(* CODESYS project proj_12_18_zad1.project

Project tree, tasks and I/O mapping:
  Device : Berghof MX6 Control, Berghof Automation GmbH, version 1.8.0.0
    application Application
      libraries: Standard, * (System)
      task MainTask (cyclic, interval t#25ms, priority 1) calls PLC_PRG
      program PLC_PRG [LD]
      visualisation Visualization
      function F_KIERUNEK [LD]
      function block FB_TIMERY [LD]
      function block FB_STER_NAPEDU [LD]
    Extension_Slots : Extension Slots, Berghof Automation GmbH, version 1.2.0.3
      XBIO_Berghof_IO : XBIO Berghof IO, Berghof Automation GmbH, version 1.2.0.3
          unmapped channels: Digital Input 0, Digital Input 1, Digital Input 2, Digital Input 3, Digital Input 4, Digital Output 0, Digital Output 1, Digital Output 2, Digital Output 3, Digital Output 4, Channel 0, Channel 1, Channel 2, Channel 3, Channel 4, Channel 5, Channel 6, Channel 7, Channel 8, Channel 9, Channel 10, Channel 11, Channel 0, Channel 1, Channel 2, Channel 3, Channel 4, Channel 5, Channel 6, Channel 7, Counter/Encoder 0, Counter/Encoder 1, Differential Counter/Encoder (0+1), DUMMY 0
      <Empty>
  text list GlobalTextList
  function block FB_STER_NAPEDU [LD]
*)

// Device/Application/PLC_PRG
PROGRAM PLC_PRG
VAR_INPUT
	CWL AT %IX0.0: BOOL;
	CWLP AT %IX0.1: BOOL;
	CWP AT %IX0.2: BOOL;
	CWPP AT %IX0.3: BOOL;
	TRASA AT %IX0.4: BOOL;
END_VAR
VAR_OUTPUT
	POD_1 AT %QX0.0: BOOL;
	POD_2 AT %QX0.1: BOOL;
	POD_3L AT %QX0.2: BOOL;
	POD_3P AT %QX0.3: BOOL;
	K1 AT %QX0.4: BOOL;
	K2 AT %QX0.5: BOOL;
END_VAR
VAR
	LICZ: CTU;
	NUM: WORD;
	FB_TIMERY_0: FB_TIMERY;
	FB_STER_NAPEDU: FB_STER_NAPEDU;
	TON1: TON;
	T1: TIME;
	FB_STER_NAPEDU_P1: FB_STER_NAPEDU;
	FB_STER_NAPEDU_P2: FB_STER_NAPEDU;
END_VAR
VAR_INPUT
	CT_RES AT %IX0.5: BOOL;
END_VAR
VAR_OUTPUT
	CT_OUT: BOOL;
END_VAR

VAR_INPUT
	ZAL_WYL_AUT_IN: BOOL;
	PRAWO_LEWO_AUT_IN: BOOL;
	ZAL_WYL_LOK_IN: BOOL;
	PRAWO_LEWO_LOK_IN: BOOL;
	POTW_ROZR_IN: BOOL;
	BLAD_ASYM_IN: BOOL;
	BLAD_TEMP_IN: BOOL;
	CHCE_LOK_IN: BOOL;
	POTW_LOK_IN: BOOL;
END_VAR

VAR_OUTPUT
	ZAL_WYL_OUT: BOOL;
	PRAWO_LEWO_OUT: BOOL;
	SYGN_OSTRZ_OUT: BOOL;
	BLAD_OUT: BOOL;
	CHCE_LOK_OUT: BOOL;
	LOK_OUT: BOOL;
	AUT_OUT: BOOL;
END_VAR
VAR_INPUT
	KASOWANIE_ALARMU: BOOL;
END_VAR
VAR
	TON0: TON;
	T0: TIME;
END_VAR
VAR_OUTPUT
	ZAL_WYL_OUT_P1: BOOL;
	ZAL_WYL_OUT_P2: BOOL;
	SYGN_OSTRZ_OUT_P1: BOOL;
	SYGN_OSTRZ_OUT_P2: BOOL;
	BLAD_OUT_P1: BOOL;
	BLAD_OUT_P2: BOOL;
	CHCE_LOK_OUT_P1: BOOL;
	CHCE_LOK_OUT_P2: BOOL;
	LOK_OUT_P1: BOOL;
	LOK_OUT_P2: BOOL;
	AUT_OUT_P1: BOOL;
	AUT_OUT_P2: BOOL;
END_VAR
VAR_INPUT
	ZAL_WYL_LOK_IN_P1: BOOL;
	ZAL_WYL_LOK_IN_P2: BOOL;
	POTW_ROZR_IN_P1: BOOL;
	POTW_ROZR_IN_P2: BOOL;
	BLAD_ASYM_IN_P1: BOOL;
	BLAD_ASYM_IN_P2: BOOL;
	BLAD_TEMP_IN_P1: BOOL;
	BLAD_TEMP_IN_P2: BOOL;
	CHCE_LOK_IN_P1: BOOL;
	CHCE_LOK_IN_P2: BOOL;
	POTW_LOK_IN_P1: BOOL;
	POTW_LOK_IN_P2: BOOL;
END_VAR
VAR
	M1: BOOL;
	M2: BOOL;
END_VAR

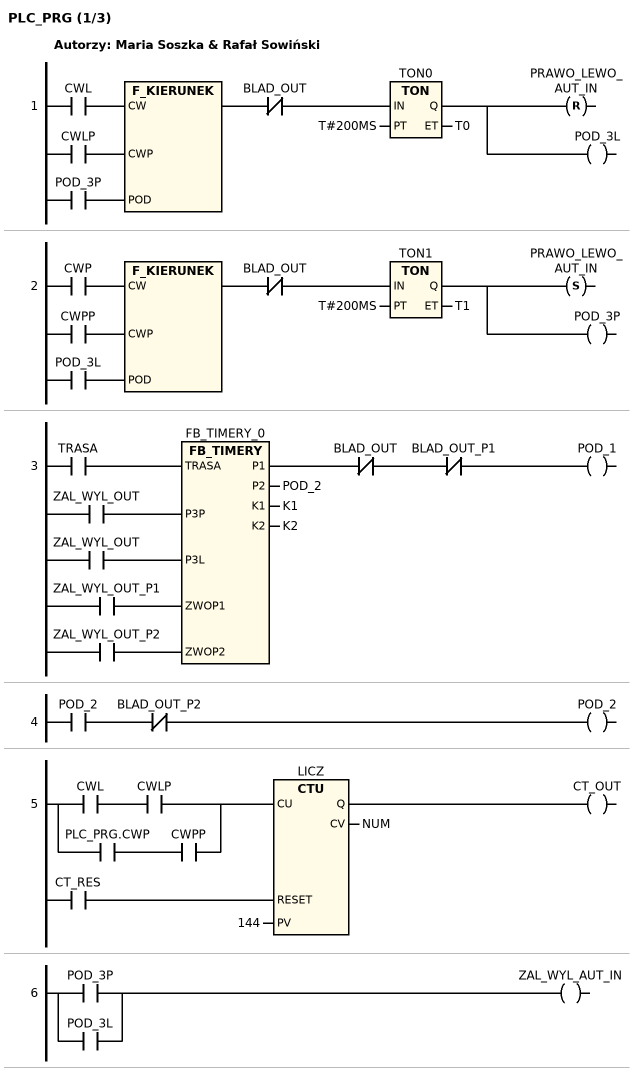
// NETWORK 1: Autorzy: Maria Soszka & Rafał Sowiński
TON0(IN := F_KIERUNEK(CW := CWL, CWP := CWLP, POD := POD_3P) AND NOT BLAD_OUT, PT := T#200MS, ET => T0); // TON
PRAWO_LEWO_AUT_IN R= TON0.Q;
POD_3L := TON0.Q;

// NETWORK 2
TON1(IN := F_KIERUNEK(CW := CWP, CWP := CWPP, POD := POD_3L) AND NOT BLAD_OUT, PT := T#200MS, ET => T1); // TON
PRAWO_LEWO_AUT_IN S= TON1.Q;
POD_3P := TON1.Q;

// NETWORK 3
FB_TIMERY_0(
    TRASA := TRASA,
    P3P := ZAL_WYL_OUT,
    P3L := ZAL_WYL_OUT,
    ZWOP1 := ZAL_WYL_OUT_P1,
    ZWOP2 := ZAL_WYL_OUT_P2,
    P2 => POD_2,
    K1 => K1,
    K2 => K2); // FB_TIMERY
POD_1 := FB_TIMERY_0.P1 AND NOT BLAD_OUT AND NOT BLAD_OUT_P1;

// NETWORK 4
POD_2 := POD_2 AND NOT BLAD_OUT_P2;

// NETWORK 5
LICZ(CU := CWL AND CWLP OR PLC_PRG.CWP AND CWPP, RESET := CT_RES, PV := 144, CV => NUM); // CTU
CT_OUT := LICZ.Q;

// NETWORK 6
ZAL_WYL_AUT_IN := POD_3P OR POD_3L;

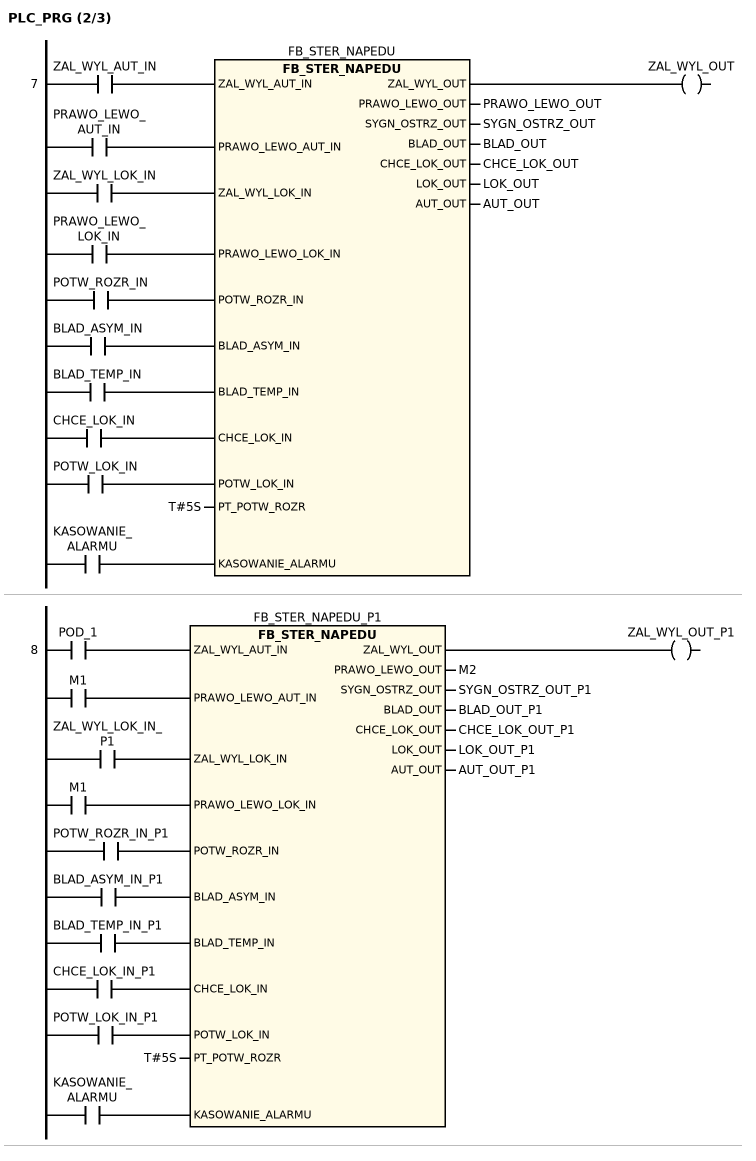
// NETWORK 7
FB_STER_NAPEDU(
    ZAL_WYL_AUT_IN := ZAL_WYL_AUT_IN,
    PRAWO_LEWO_AUT_IN := PRAWO_LEWO_AUT_IN,
    ZAL_WYL_LOK_IN := ZAL_WYL_LOK_IN,
    PRAWO_LEWO_LOK_IN := PRAWO_LEWO_LOK_IN,
    POTW_ROZR_IN := POTW_ROZR_IN,
    BLAD_ASYM_IN := BLAD_ASYM_IN,
    BLAD_TEMP_IN := BLAD_TEMP_IN,
    CHCE_LOK_IN := CHCE_LOK_IN,
    POTW_LOK_IN := POTW_LOK_IN,
    PT_POTW_ROZR := T#5S,
    KASOWANIE_ALARMU := KASOWANIE_ALARMU,
    PRAWO_LEWO_OUT => PRAWO_LEWO_OUT,
    SYGN_OSTRZ_OUT => SYGN_OSTRZ_OUT,
    BLAD_OUT => BLAD_OUT,
    CHCE_LOK_OUT => CHCE_LOK_OUT,
    LOK_OUT => LOK_OUT,
    AUT_OUT => AUT_OUT);
ZAL_WYL_OUT := FB_STER_NAPEDU.ZAL_WYL_OUT;

// NETWORK 8
FB_STER_NAPEDU_P1(
    ZAL_WYL_AUT_IN := POD_1,
    PRAWO_LEWO_AUT_IN := M1,
    ZAL_WYL_LOK_IN := ZAL_WYL_LOK_IN_P1,
    PRAWO_LEWO_LOK_IN := M1,
    POTW_ROZR_IN := POTW_ROZR_IN_P1,
    BLAD_ASYM_IN := BLAD_ASYM_IN_P1,
    BLAD_TEMP_IN := BLAD_TEMP_IN_P1,
    CHCE_LOK_IN := CHCE_LOK_IN_P1,
    POTW_LOK_IN := POTW_LOK_IN_P1,
    PT_POTW_ROZR := T#5S,
    KASOWANIE_ALARMU := KASOWANIE_ALARMU,
    PRAWO_LEWO_OUT => M2,
    SYGN_OSTRZ_OUT => SYGN_OSTRZ_OUT_P1,
    BLAD_OUT => BLAD_OUT_P1,
    CHCE_LOK_OUT => CHCE_LOK_OUT_P1,
    LOK_OUT => LOK_OUT_P1,
    AUT_OUT => AUT_OUT_P1); // FB_STER_NAPEDU
ZAL_WYL_OUT_P1 := FB_STER_NAPEDU_P1.ZAL_WYL_OUT;

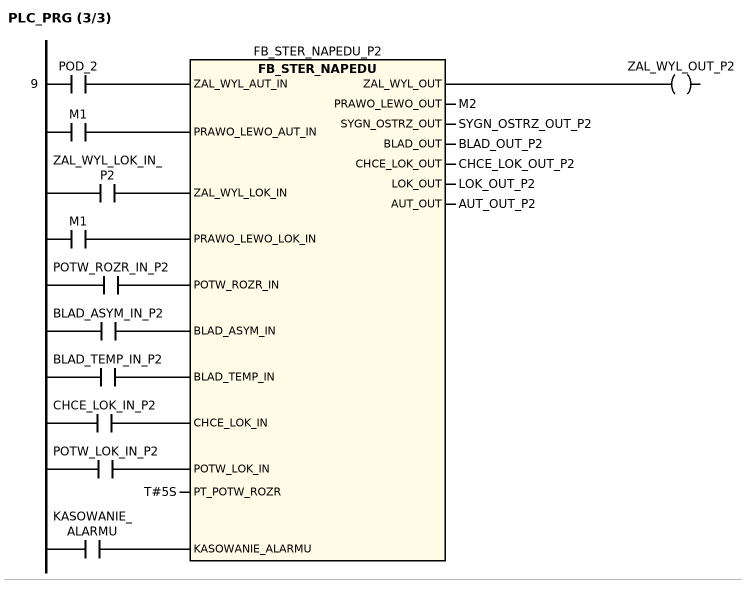
// NETWORK 9
FB_STER_NAPEDU_P2(
    ZAL_WYL_AUT_IN := POD_2,
    PRAWO_LEWO_AUT_IN := M1,
    ZAL_WYL_LOK_IN := ZAL_WYL_LOK_IN_P2,
    PRAWO_LEWO_LOK_IN := M1,
    POTW_ROZR_IN := POTW_ROZR_IN_P2,
    BLAD_ASYM_IN := BLAD_ASYM_IN_P2,
    BLAD_TEMP_IN := BLAD_TEMP_IN_P2,
    CHCE_LOK_IN := CHCE_LOK_IN_P2,
    POTW_LOK_IN := POTW_LOK_IN_P2,
    PT_POTW_ROZR := T#5S,
    KASOWANIE_ALARMU := KASOWANIE_ALARMU,
    PRAWO_LEWO_OUT => M2,
    SYGN_OSTRZ_OUT => SYGN_OSTRZ_OUT_P2,
    BLAD_OUT => BLAD_OUT_P2,
    CHCE_LOK_OUT => CHCE_LOK_OUT_P2,
    LOK_OUT => LOK_OUT_P2,
    AUT_OUT => AUT_OUT_P2); // FB_STER_NAPEDU
ZAL_WYL_OUT_P2 := FB_STER_NAPEDU_P2.ZAL_WYL_OUT;

END_PROGRAM

// Device/Application/F_KIERUNEK
FUNCTION F_KIERUNEK : BOOL
VAR_INPUT
	CW: BOOL;
	CWP: BOOL;
	POD: BOOL;
END_VAR

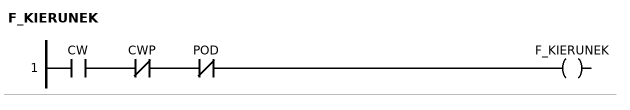
// NETWORK 1
F_KIERUNEK := CW AND NOT CWP AND NOT POD;

END_FUNCTION

// Device/Application/FB_TIMERY
FUNCTION_BLOCK FB_TIMERY
VAR_INPUT
	TRASA: BOOL;
END_VAR
VAR_OUTPUT
	P1: BOOL;
	P2: BOOL;
	K1: BOOL;
	K2: BOOL;
END_VAR
VAR
	TIM1: TON;
	T1: TIME;
	TIM2: TON;
	T2: TIME;
	TIMK1: TON;
	TIMK2: TON;
	TK1: TIME;
	TK2: TIME;
END_VAR
VAR_INPUT
	P3P: BOOL;
	P3L: BOOL;
	ZWOP1: BOOL;
	ZWOP2: BOOL;
END_VAR
VAR // added by the converter: edge detectors and wires of the graphical bodies
    _w1 : BOOL;
END_VAR

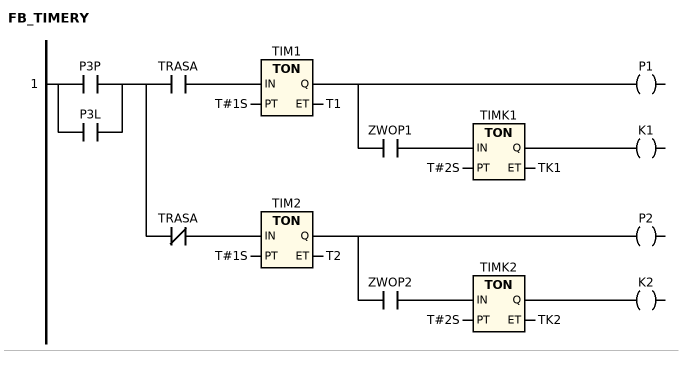
// NETWORK 1
_w1 := P3P OR P3L;
TIM1(IN := _w1 AND TRASA, PT := T#1S, ET => T1); // TON
P1 := TIM1.Q;
TIMK1(IN := TIM1.Q AND ZWOP1, PT := T#2S, ET => TK1); // TON
K1 := TIMK1.Q;
TIM2(IN := _w1 AND NOT TRASA, PT := T#1S, ET => T2); // TON
P2 := TIM2.Q;
TIMK2(IN := TIM2.Q AND ZWOP2, PT := T#2S, ET => TK2); // TON
K2 := TIMK2.Q;

END_FUNCTION_BLOCK

// FB_STER_NAPEDU
FUNCTION_BLOCK FB_STER_NAPEDU
VAR_INPUT
	ZAL_WYL_AUT_IN: BOOL;
	PRAWO_LEWO_AUT_IN: BOOL;
	ZAL_WYL_LOK_IN: BOOL;
	PRAWO_LEWO_LOK_IN: BOOL;
	POTW_ROZR_IN: BOOL;
	BLAD_ASYM_IN: BOOL;
	BLAD_TEMP_IN: BOOL;
	CHCE_LOK_IN: BOOL;
	POTW_LOK_IN: BOOL;
END_VAR
VAR_OUTPUT
	ZAL_WYL_OUT: BOOL;
	PRAWO_LEWO_OUT: BOOL;
	SYGN_OSTRZ_OUT: BOOL;
	BLAD_OUT: BOOL;
	CHCE_LOK_OUT: BOOL;
	LOK_OUT: BOOL;
	AUT_OUT: BOOL;
END_VAR
VAR
	BRAK_POTW_ROZR: BOOL;
	TON_SYGN_OSTRZ: TON;
	T_SYGN_OSTRZ: TIME;
	PT_SYGN_OSTRZ: TIME := T#3S;
	TON_POTW_ROZR: TON;
	T_POTW_ROZR: TIME;
END_VAR
VAR_INPUT
	PT_POTW_ROZR: TIME;
END_VAR
VAR // added by the converter: edge detectors and wires of the graphical bodies
    _w1 : BOOL;
END_VAR

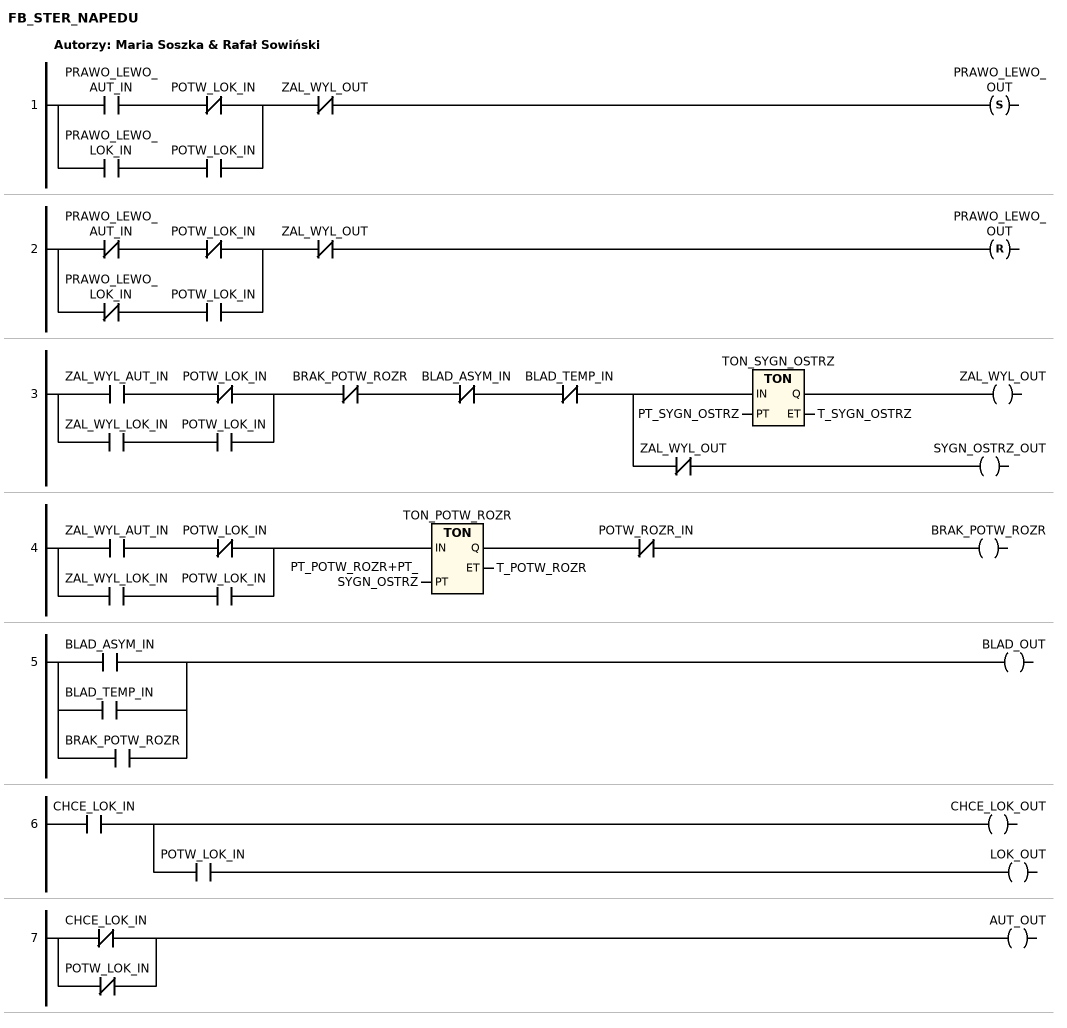
// NETWORK 1: Autorzy: Maria Soszka & Rafał Sowiński
PRAWO_LEWO_OUT S= (PRAWO_LEWO_AUT_IN AND NOT POTW_LOK_IN OR PRAWO_LEWO_LOK_IN AND POTW_LOK_IN) AND NOT ZAL_WYL_OUT;

// NETWORK 2
PRAWO_LEWO_OUT R= (NOT PRAWO_LEWO_AUT_IN AND NOT POTW_LOK_IN OR NOT PRAWO_LEWO_LOK_IN AND POTW_LOK_IN) AND NOT ZAL_WYL_OUT;

// NETWORK 3
_w1 := (ZAL_WYL_AUT_IN AND NOT POTW_LOK_IN OR ZAL_WYL_LOK_IN AND POTW_LOK_IN) AND NOT BRAK_POTW_ROZR AND NOT BLAD_ASYM_IN AND NOT BLAD_TEMP_IN;
TON_SYGN_OSTRZ(IN := _w1, PT := PT_SYGN_OSTRZ, ET => T_SYGN_OSTRZ); // TON
ZAL_WYL_OUT := TON_SYGN_OSTRZ.Q;
SYGN_OSTRZ_OUT := _w1 AND NOT ZAL_WYL_OUT;

// NETWORK 4
TON_POTW_ROZR(
    IN := ZAL_WYL_AUT_IN AND NOT POTW_LOK_IN OR ZAL_WYL_LOK_IN AND POTW_LOK_IN,
    PT := PT_POTW_ROZR+PT_SYGN_OSTRZ,
    ET => T_POTW_ROZR); // TON
BRAK_POTW_ROZR := TON_POTW_ROZR.Q AND NOT POTW_ROZR_IN;

// NETWORK 5
BLAD_OUT := BLAD_ASYM_IN OR BLAD_TEMP_IN OR BRAK_POTW_ROZR;

// NETWORK 6
CHCE_LOK_OUT := CHCE_LOK_IN;
LOK_OUT := CHCE_LOK_IN AND POTW_LOK_IN;

// NETWORK 7
AUT_OUT := NOT CHCE_LOK_IN OR NOT POTW_LOK_IN;

END_FUNCTION_BLOCK

// Device/Application/FB_STER_NAPEDU
FUNCTION_BLOCK FB_STER_NAPEDU
VAR_INPUT
	ZAL_WYL_AUT_IN: BOOL;
	PRAWO_LEWO_AUT_IN: BOOL;
	ZAL_WYL_LOK_IN: BOOL;
	PRAWO_LEWO_LOK_IN: BOOL;
	POTW_ROZR_IN: BOOL;
	BLAD_ASYM_IN: BOOL;
	BLAD_TEMP_IN: BOOL;
	CHCE_LOK_IN: BOOL;
	POTW_LOK_IN: BOOL;
END_VAR
VAR_OUTPUT
	ZAL_WYL_OUT: BOOL;
	PRAWO_LEWO_OUT: BOOL;
	SYGN_OSTRZ_OUT: BOOL;
	BLAD_OUT: BOOL;
	CHCE_LOK_OUT: BOOL;
	LOK_OUT: BOOL;
	AUT_OUT: BOOL;
END_VAR
VAR
	BRAK_POTW_ROZR: BOOL;
	TON_SYGN_OSTRZ: TON;
	T_SYGN_OSTRZ: TIME;
	PT_SYGN_OSTRZ: TIME := T#3S;
	TON_POTW_ROZR: TON;
	T_POTW_ROZR: TIME;
END_VAR
VAR_INPUT
	PT_POTW_ROZR: TIME;
	KASOWANIE_ALARMU: BOOL;
END_VAR
VAR // added by the converter: edge detectors and wires of the graphical bodies
    _w1 : BOOL;
END_VAR

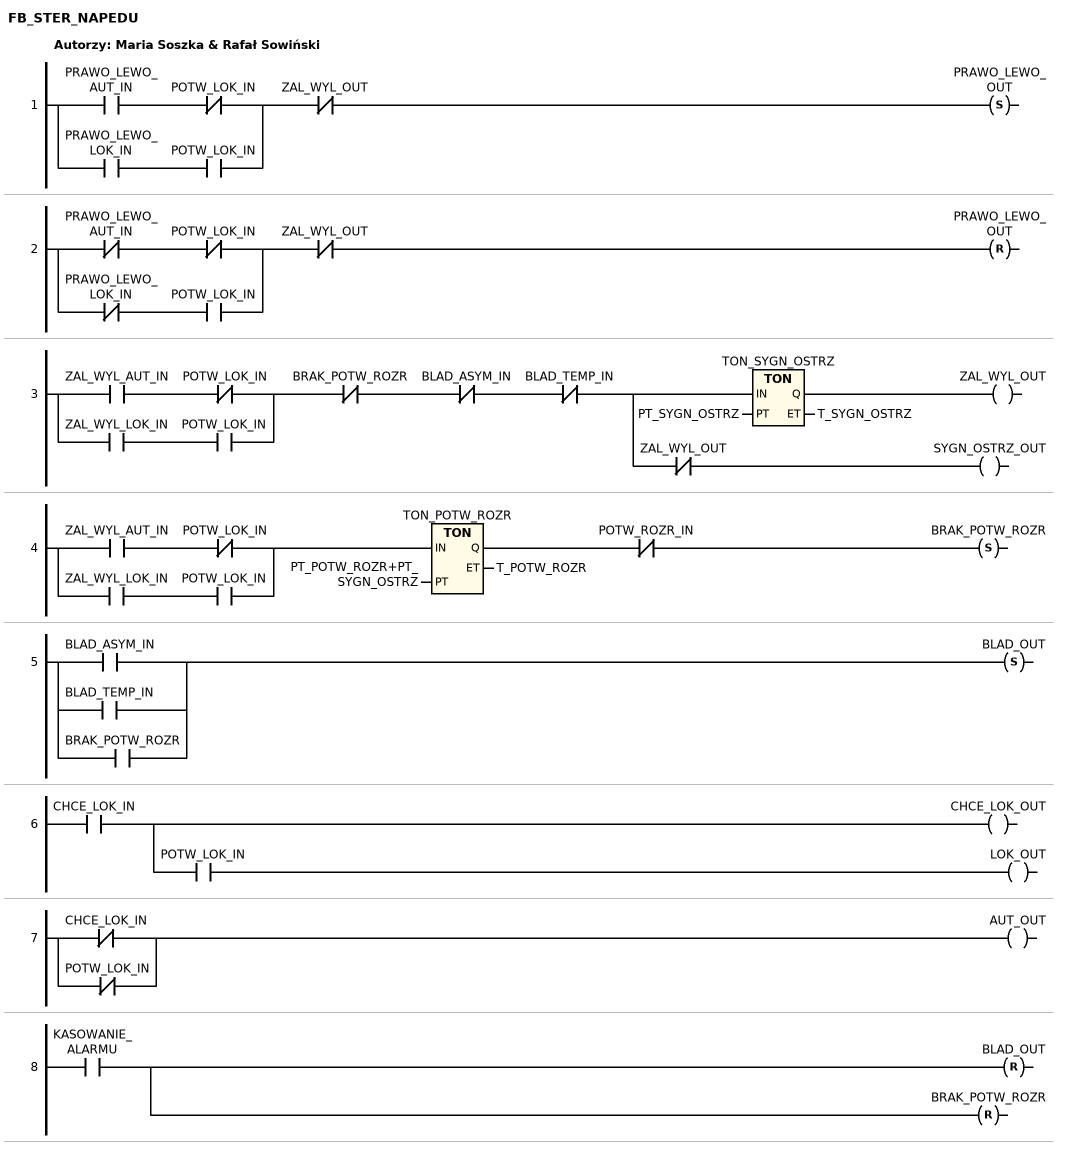
// NETWORK 1: Autorzy: Maria Soszka & Rafał Sowiński
PRAWO_LEWO_OUT S= (PRAWO_LEWO_AUT_IN AND NOT POTW_LOK_IN OR PRAWO_LEWO_LOK_IN AND POTW_LOK_IN) AND NOT ZAL_WYL_OUT;

// NETWORK 2
PRAWO_LEWO_OUT R= (NOT PRAWO_LEWO_AUT_IN AND NOT POTW_LOK_IN OR NOT PRAWO_LEWO_LOK_IN AND POTW_LOK_IN) AND NOT ZAL_WYL_OUT;

// NETWORK 3
_w1 := (ZAL_WYL_AUT_IN AND NOT POTW_LOK_IN OR ZAL_WYL_LOK_IN AND POTW_LOK_IN) AND NOT BRAK_POTW_ROZR AND NOT BLAD_ASYM_IN AND NOT BLAD_TEMP_IN;
TON_SYGN_OSTRZ(IN := _w1, PT := PT_SYGN_OSTRZ, ET => T_SYGN_OSTRZ); // TON
ZAL_WYL_OUT := TON_SYGN_OSTRZ.Q;
SYGN_OSTRZ_OUT := _w1 AND NOT ZAL_WYL_OUT;

// NETWORK 4
TON_POTW_ROZR(
    IN := ZAL_WYL_AUT_IN AND NOT POTW_LOK_IN OR ZAL_WYL_LOK_IN AND POTW_LOK_IN,
    PT := PT_POTW_ROZR+PT_SYGN_OSTRZ,
    ET => T_POTW_ROZR); // TON
BRAK_POTW_ROZR S= TON_POTW_ROZR.Q AND NOT POTW_ROZR_IN;

// NETWORK 5
BLAD_OUT S= BLAD_ASYM_IN OR BLAD_TEMP_IN OR BRAK_POTW_ROZR;

// NETWORK 6
CHCE_LOK_OUT := CHCE_LOK_IN;
LOK_OUT := CHCE_LOK_IN AND POTW_LOK_IN;

// NETWORK 7
AUT_OUT := NOT CHCE_LOK_IN OR NOT POTW_LOK_IN;

// NETWORK 8
BLAD_OUT R= KASOWANIE_ALARMU;
BRAK_POTW_ROZR R= KASOWANIE_ALARMU;

END_FUNCTION_BLOCK

// Device/Application/Visualization
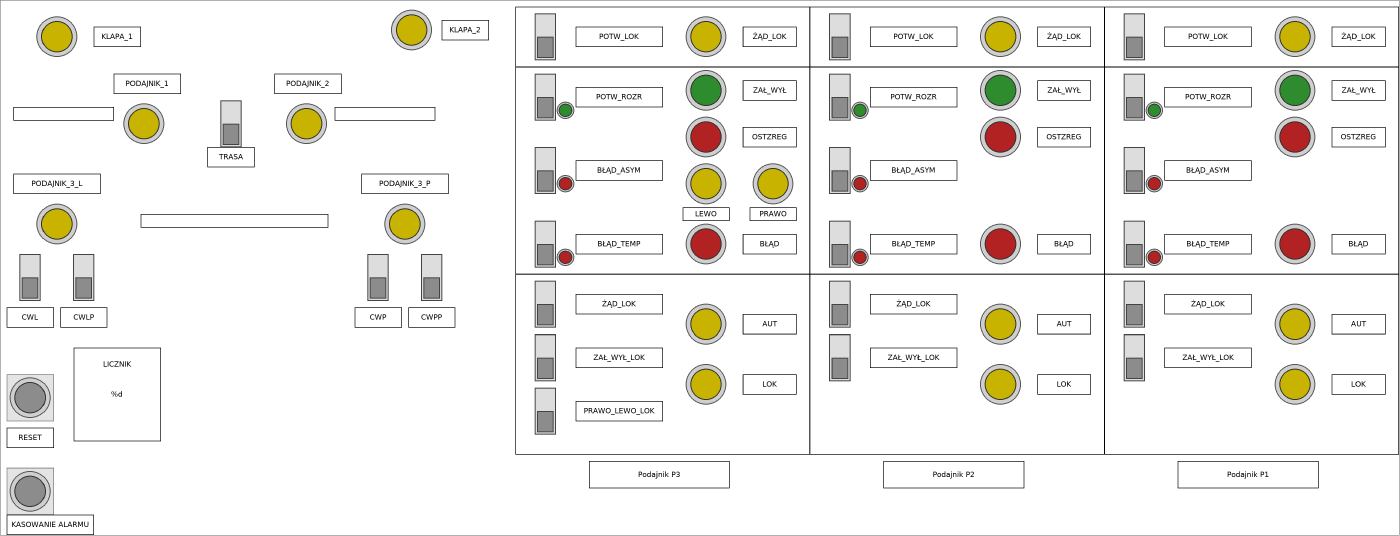
VISUALIZATION Visualization  // 2092x802
    DipSwitch (10,380 70x70), variable: PLC_PRG.CWL, behaviour: TOGGLE, style: Switch-DipSwitch-Gray
    DipSwitch (90,380 70x70), variable: PLC_PRG.CWLP, behaviour: TOGGLE, style: Switch-DipSwitch-Gray
    DipSwitch (530,380 70x70), variable: PLC_PRG.CWP, behaviour: TOGGLE, style: Switch-DipSwitch-Gray
    DipSwitch (610,380 70x70), variable: PLC_PRG.CWPP, behaviour: TOGGLE, style: Switch-DipSwitch-Gray
    PushSwitch (10,560 70x70), variable: PLC_PRG.CT_RES, behaviour: TAP, style: Switch-PushSwitch-Gray
    Lamp1 (570,300 70x70), variable: PLC_PRG.PRAWO_LEWO_OUT, style: Lamp-Lamp1-Yellow
    Lamp1 (50,300 70x70), variable: NOT PLC_PRG.PRAWO_LEWO_OUT, style: Lamp-Lamp1-Yellow
    Lamp1 (423,150 70x70), variable: PLC_PRG.ZAL_WYL_OUT_P2, style: Lamp-Lamp1-Yellow
    Lamp1 (180,150 70x70), variable: PLC_PRG.ZAL_WYL_OUT_P1, style: Lamp-Lamp1-Yellow
    DipSwitch (310,150 70x70), variable: PLC_PRG.TRASA, behaviour: TOGGLE, style: Switch-DipSwitch-Gray
    Lamp1 (50,20 70x70), variable: PLC_PRG.K1, style: Lamp-Lamp1-Yellow
    Lamp1 (580,10 70x70), variable: PLC_PRG.K2, style: Lamp-Lamp1-Yellow
    RoundedRectangle (110,520 130x140), "%d", text variable: PLC_PRG.NUM
    Label (100,530 150x30), "LICZNIK"
    RoundedRectangle (530,460 70x30)
    RoundedRectangle (610,460 70x30)
    Label (500,450 130x50), "CWP"
    Label (600,440 90x70), "CWPP"
    RoundedRectangle (10,460 70x30), "CWL"
    RoundedRectangle (90,460 70x30), "CWLP"
    RoundedRectangle (310,220 70x30), "TRASA"
    RoundedRectangle (540,260 130x30), "PODAJNIK_3_P"
    RoundedRectangle (20,260 130x30), "PODAJNIK_3_L"
    RoundedRectangle (170,110 100x30), "PODAJNIK_1"
    RoundedRectangle (410,110 100x30), "PODAJNIK_2"
    RoundedRectangle (660,30 70x30), "KLAPA_2"
    RoundedRectangle (140,40 70x30), "KLAPA_1"
    RoundedRectangle (10,640 70x30), "RESET"
    Rectangle (210,320 280x20), colour toggle: PLC_PRG.ZAL_WYL_OUT
    Rectangle (500,160 150x20), colour toggle: PLC_PRG.ZAL_WYL_OUT_P2
    Rectangle (20,160 150x20), colour toggle: PLC_PRG.ZAL_WYL_OUT_P1
    Rectangle (770,410 440x270)
    Rectangle (770,100 440x310)
    DipSwitch (780,110 70x70), variable: PLC_PRG.POTW_ROZR_IN, behaviour: TOGGLE, style: Switch-DipSwitch-Gray
    Rectangle (770,10 440x90)
    DipSwitch (780,220 70x70), variable: PLC_PRG.BLAD_ASYM_IN, behaviour: TOGGLE, style: Switch-DipSwitch-Gray
    DipSwitch (780,330 70x70), variable: PLC_PRG.BLAD_TEMP_IN, behaviour: TOGGLE, style: Switch-DipSwitch-Gray
    DipSwitch (780,500 70x70), variable: PLC_PRG.ZAL_WYL_LOK_IN, behaviour: TOGGLE, style: Switch-DipSwitch-Gray
    DipSwitch (780,420 70x70), variable: PLC_PRG.CHCE_LOK_IN, behaviour: TOGGLE, style: Switch-DipSwitch-Gray
    DipSwitch (780,580 70x70), variable: PLC_PRG.PRAWO_LEWO_LOK_IN, behaviour: TOGGLE, style: Switch-DipSwitch-Gray
    Lamp1 (1020,20 70x70), variable: PLC_PRG.CHCE_LOK_OUT, style: Lamp-Lamp1-Yellow
    Lamp1 (1020,100 70x70), variable: PLC_PRG.ZAL_WYL_OUT, style: Lamp-Lamp1-Green
    Lamp1 (1020,240 70x70), variable: NOT PLC_PRG.PRAWO_LEWO_OUT, style: Lamp-Lamp1-Yellow
    Lamp1 (1020,170 70x70), variable: PLC_PRG.SYGN_OSTRZ_OUT, style: Lamp-Lamp1-Red
    Lamp1 (1120,240 70x70), variable: PLC_PRG.PRAWO_LEWO_OUT, style: Lamp-Lamp1-Yellow
    Lamp1 (1020,450 70x70), variable: PLC_PRG.AUT_OUT, style: Lamp-Lamp1-Yellow
    Lamp1 (1020,540 70x70), variable: PLC_PRG.LOK_OUT, style: Lamp-Lamp1-Yellow
    Lamp1 (1020,330 70x70), variable: PLC_PRG.BLAD_OUT, style: Lamp-Lamp1-Red
    Rectangle (860,40 130x30), "POTW_LOK"
    Rectangle (1110,40 80x30), "ŻĄD_LOK"
    Rectangle (860,130 130x30), "POTW_ROZR"
    Rectangle (860,240 130x30), "BŁĄD_ASYM"
    Rectangle (860,350 130x30), "BŁĄD_TEMP"
    Rectangle (1020,310 70x20), "LEWO"
    Rectangle (1120,310 70x20), "PRAWO"
    Rectangle (1110,120 80x30), "ZAŁ_WYŁ"
    Rectangle (1110,190 80x30), "OSTZREG"
    Rectangle (1110,350 80x30), "BŁĄD"
    Rectangle (860,440 130x30), "ŻĄD_LOK"
    Rectangle (860,520 130x30), "ZAŁ_WYŁ_LOK"
    Rectangle (860,600 130x30), "PRAWO_LEWO_LOK"
    Rectangle (1110,470 80x30), "AUT"
    Rectangle (1110,560 80x30), "LOK"
    DipSwitch (780,20 70x70), variable: PLC_PRG.POTW_LOK_IN, behaviour: TOGGLE, style: Switch-DipSwitch-Gray
    Lamp1 (830,150 30x30), variable: PLC_PRG.POTW_ROZR_IN, style: Lamp-Lamp1-Green
    Lamp1 (830,260 30x30), variable: PLC_PRG.BLAD_ASYM_IN, style: Lamp-Lamp1-Red
    Lamp1 (830,370 30x30), variable: PLC_PRG.BLAD_TEMP_IN, style: Lamp-Lamp1-Red
    PushSwitch (10,700 70x70), variable: PLC_PRG.KASOWANIE_ALARMU, behaviour: TAP, style: Switch-PushSwitch-Gray
    Rectangle (10,770 130x30), "KASOWANIE ALARMU"
    Rectangle (1210,410 440x270)
    Rectangle (1210,100 440x310)
    DipSwitch (1220,110 70x70), variable: PLC_PRG.POTW_ROZR_IN_P2, behaviour: TOGGLE, style: Switch-DipSwitch-Gray
    Rectangle (1210,10 440x90)
    DipSwitch (1220,220 70x70), variable: PLC_PRG.BLAD_ASYM_IN_P2, behaviour: TOGGLE, style: Switch-DipSwitch-Gray
    DipSwitch (1220,330 70x70), variable: PLC_PRG.BLAD_TEMP_IN_P2, behaviour: TOGGLE, style: Switch-DipSwitch-Gray
    DipSwitch (1220,500 70x70), variable: PLC_PRG.ZAL_WYL_LOK_IN_P2, behaviour: TOGGLE, style: Switch-DipSwitch-Gray
    DipSwitch (1220,420 70x70), variable: PLC_PRG.CHCE_LOK_IN_P2, behaviour: TOGGLE, style: Switch-DipSwitch-Gray
    Lamp1 (1460,20 70x70), variable: PLC_PRG.CHCE_LOK_OUT_P2, style: Lamp-Lamp1-Yellow
    Lamp1 (1460,100 70x70), variable: PLC_PRG.ZAL_WYL_OUT_P2, style: Lamp-Lamp1-Green
    Lamp1 (1460,170 70x70), variable: PLC_PRG.SYGN_OSTRZ_OUT_P2, style: Lamp-Lamp1-Red
    Lamp1 (1460,450 70x70), variable: PLC_PRG.AUT_OUT_P2, style: Lamp-Lamp1-Yellow
    Lamp1 (1460,540 70x70), variable: PLC_PRG.LOK_OUT_P2, style: Lamp-Lamp1-Yellow
    Lamp1 (1460,330 70x70), variable: PLC_PRG.BLAD_OUT_P2, style: Lamp-Lamp1-Red
    Rectangle (1300,40 130x30), "POTW_LOK"
    Rectangle (1550,40 80x30), "ŻĄD_LOK"
    Rectangle (1300,130 130x30), "POTW_ROZR"
    Rectangle (1300,240 130x30), "BŁĄD_ASYM"
    Rectangle (1300,350 130x30), "BŁĄD_TEMP"
    Rectangle (1550,120 80x30), "ZAŁ_WYŁ"
    Rectangle (1550,190 80x30), "OSTZREG"
    Rectangle (1550,350 80x30), "BŁĄD"
    Rectangle (1300,440 130x30), "ŻĄD_LOK"
    Rectangle (1300,520 130x30), "ZAŁ_WYŁ_LOK"
    Rectangle (1550,470 80x30), "AUT"
    Rectangle (1550,560 80x30), "LOK"
    DipSwitch (1220,20 70x70), variable: PLC_PRG.POTW_LOK_IN_P2, behaviour: TOGGLE, style: Switch-DipSwitch-Gray
    Lamp1 (1270,150 30x30), variable: PLC_PRG.POTW_ROZR_IN_P2, style: Lamp-Lamp1-Green
    Lamp1 (1270,260 30x30), variable: PLC_PRG.BLAD_ASYM_IN_P2, style: Lamp-Lamp1-Red
    Lamp1 (1270,370 30x30), variable: PLC_PRG.BLAD_TEMP_IN_P2, style: Lamp-Lamp1-Red
    Rectangle (1650,410 440x270)
    Rectangle (1650,100 440x310)
    DipSwitch (1660,110 70x70), variable: PLC_PRG.POTW_ROZR_IN_P1, behaviour: TOGGLE, style: Switch-DipSwitch-Gray
    Rectangle (1650,10 440x90)
    DipSwitch (1660,220 70x70), variable: PLC_PRG.BLAD_ASYM_IN_P1, behaviour: TOGGLE, style: Switch-DipSwitch-Gray
    DipSwitch (1660,330 70x70), variable: PLC_PRG.BLAD_TEMP_IN_P1, behaviour: TOGGLE, style: Switch-DipSwitch-Gray
    DipSwitch (1660,500 70x70), variable: PLC_PRG.ZAL_WYL_LOK_IN_P1, behaviour: TOGGLE, style: Switch-DipSwitch-Gray
    DipSwitch (1660,420 70x70), variable: PLC_PRG.CHCE_LOK_IN_P1, behaviour: TOGGLE, style: Switch-DipSwitch-Gray
    Lamp1 (1900,20 70x70), variable: PLC_PRG.CHCE_LOK_OUT_P1, style: Lamp-Lamp1-Yellow
    Lamp1 (1900,100 70x70), variable: PLC_PRG.ZAL_WYL_OUT_P1, style: Lamp-Lamp1-Green
    Lamp1 (1900,170 70x70), variable: PLC_PRG.SYGN_OSTRZ_OUT_P1, style: Lamp-Lamp1-Red
    Lamp1 (1900,450 70x70), variable: PLC_PRG.AUT_OUT_P1, style: Lamp-Lamp1-Yellow
    Lamp1 (1900,540 70x70), variable: PLC_PRG.LOK_OUT_P1, style: Lamp-Lamp1-Yellow
    Lamp1 (1900,330 70x70), variable: PLC_PRG.BLAD_OUT_P1, style: Lamp-Lamp1-Red
    Rectangle (1740,40 130x30), "POTW_LOK"
    Rectangle (1990,40 80x30), "ŻĄD_LOK"
    Rectangle (1740,130 130x30), "POTW_ROZR"
    Rectangle (1740,240 130x30), "BŁĄD_ASYM"
    Rectangle (1740,350 130x30), "BŁĄD_TEMP"
    Rectangle (1990,120 80x30), "ZAŁ_WYŁ"
    Rectangle (1990,190 80x30), "OSTZREG"
    Rectangle (1990,350 80x30), "BŁĄD"
    Rectangle (1740,440 130x30), "ŻĄD_LOK"
    Rectangle (1740,520 130x30), "ZAŁ_WYŁ_LOK"
    Rectangle (1990,470 80x30), "AUT"
    Rectangle (1990,560 80x30), "LOK"
    DipSwitch (1660,20 70x70), variable: PLC_PRG.POTW_LOK_IN_P1, behaviour: TOGGLE, style: Switch-DipSwitch-Gray
    Lamp1 (1710,150 30x30), variable: PLC_PRG.POTW_ROZR_IN_P1, style: Lamp-Lamp1-Green
    Lamp1 (1710,260 30x30), variable: PLC_PRG.BLAD_ASYM_IN_P1, style: Lamp-Lamp1-Red
    Lamp1 (1710,370 30x30), variable: PLC_PRG.BLAD_TEMP_IN_P1, style: Lamp-Lamp1-Red
    Rectangle (880,690 210x40), "Podajnik P3"
    Rectangle (1320,690 210x40), "Podajnik P2"
    Rectangle (1760,690 210x40), "Podajnik P1"
END_VISUALIZATION
